// TIA Portal V20 export
DATA_BLOCK "Alarms"   // DB38
{ DB_Accessible_From_OPC_UA := 'FALSE' }
AUTHOR : ERsystem_FA2_DH. Kim
// stored: DBAccessibleFromOPCUA false, DBAccessibleFromWebserver false, MemoryReserve 100, Namespace Unit1.Em6
   VAR
      emAlarms { ExternalWritable := 'False'} : "LAF_typeAlarms";
      maintenanceFaults { ExternalWritable := 'False'} : Array[0..199] of Bool;   // PFE Maintenance Faults
      productionFaults { ExternalWritable := 'False'} : Array[0..199] of Bool;   // PFE Production Faults
      toolingFault { ExternalWritable := 'False'} : Array[0..199] of Bool;   // PFE Tooling Faults
      qualityFault { ExternalWritable := 'False'} : Array[0..199] of Bool;   // PFE Quality Faults
      throughputFaultBlocked { ExternalWritable := 'False'} : Array[0..199] of Bool;   // PFE Throughput Fault Blocked
      throughputFaultStarved { ExternalWritable := 'False'} : Array[0..199] of Bool;   // PFE Throughput Fault Starved
      throughputFault { ExternalWritable := 'False'} : Array[0..199] of Bool;   // PFE Throughput Fault
      systemFaultGeneral { ExternalWritable := 'False'} : Array[0..199] of Bool;   // PFE System Fault General
      materialFault { ExternalWritable := 'False'} : Array[0..199] of Bool;   // PFE Material Fault
      maintenanceWarnings { ExternalWritable := 'False'} : Array[0..199] of Bool;   // PFE Maintenance Warnings
      productionWarning { ExternalWritable := 'False'} : Array[0..199] of Bool;   // PFE Production Warning
      toolingWarning { ExternalWritable := 'False'} : Array[0..199] of Bool;   // PFE Tooling Warning
      qualityWarning { ExternalWritable := 'False'} : Array[0..199] of Bool;   // PFE Quality Warning
      throughputWarning { ExternalWritable := 'False'} : Array[0..199] of Bool;   // PFE Throughput Warning
      systemWarning { ExternalWritable := 'False'} : Array[0..199] of Bool;   // PFE System Warning
      materialWarning { ExternalWritable := 'False'} : Array[0..199] of Bool;   // PFE Material Warning
      maintenanceStatus { ExternalWritable := 'False'} : Array[0..199] of Bool;   // PFE Maintenance Status
      productionStatus { ExternalWritable := 'False'} : Array[0..199] of Bool;   // PFE Production Status
      toolingStatus { ExternalWritable := 'False'} : Array[0..199] of Bool;   // PFE Tooling Status
      qualityStatus { ExternalWritable := 'False'} : Array[0..199] of Bool;   // PFE Quality Status
      throughputStatus { ExternalWritable := 'False'} : Array[0..199] of Bool;   // PFE Throughput Status
      systemStatus { ExternalWritable := 'False'} : Array[0..199] of Bool;   // PFE System Status
      materialStatus { ExternalWritable := 'False'} : Array[0..199] of Bool;   // PFE Material Status
      tonMaintenanceFault { ExternalWritable := 'False'} : Array[0..199] of TON_TIME;   // PFE Maintenance Faults Ton Timer
      tonProductionFault { ExternalWritable := 'False'} : Array[0..199] of TON_TIME;   // PFE Production Faults Ton Timer
      tonToolingFault { ExternalWritable := 'False'} : Array[0..199] of TON_TIME;   // PFE Tooling Faults Ton Timer
      tonQualityFault { ExternalWritable := 'False'} : Array[0..199] of TON_TIME;   // PFE Quality Faults Ton Timer
      tonThroughputFaultBlocked { ExternalWritable := 'False'} : Array[0..199] of TON_TIME;   // PFE Throughput Fault Blocked Ton Timer
      tonThroughputFaultStarved { ExternalWritable := 'False'} : Array[0..199] of TON_TIME;   // PFE Throughput Fault Starved Ton Timer
      tonThroughputFault { ExternalWritable := 'False'} : Array[0..199] of TON_TIME;   // PFE Throughput Fault Ton Timer
      tonSystemFaultGeneral { ExternalWritable := 'False'} : Array[0..199] of TON_TIME;   // PFE System Fault General Ton Timer
      tonMaterialFault { ExternalWritable := 'False'} : Array[0..199] of TON_TIME;   // PFE Material Fault Ton Timer
      tonMaintenanceWarning { ExternalWritable := 'False'} : Array[0..199] of TON_TIME;   // PFE Maintenance Warnings Ton Timer
      tonProductionWarning { ExternalWritable := 'False'} : Array[0..199] of TON_TIME;   // PFE Production Warning Ton Timer
      tonToolingWarning { ExternalWritable := 'False'} : Array[0..199] of TON_TIME;   // PFE Tooling Warning Ton Timer
      tonQualityWarning { ExternalWritable := 'False'} : Array[0..199] of TON_TIME;   // PFE Quality Warning Ton Timer
      tonThroughputWarning { ExternalWritable := 'False'} : Array[0..199] of TON_TIME;   // PFE Throughput Warning Ton Timer
      tonSystemWarning { ExternalWritable := 'False'} : Array[0..199] of TON_TIME;   // PFE System Warning Ton Timer
      tonMaterialWarning { ExternalWritable := 'False'} : Array[0..199] of TON_TIME;   // PFE Material Warning Ton Timer
      tonMaintenanceStatus { ExternalWritable := 'False'} : Array[0..199] of TON_TIME;   // PFE Maintenance Status Ton Timer
      tonProductionStatus { ExternalWritable := 'False'} : Array[0..199] of TON_TIME;   // PFE Production Status Ton Timer
      tonToolingStatus { ExternalWritable := 'False'} : Array[0..199] of TON_TIME;   // PFE Tooling Status Ton Timer
      tonQualityStatus { ExternalWritable := 'False'} : Array[0..199] of TON_TIME;   // PFE Quality Status Ton Timer
      tonThroughputStatus { ExternalWritable := 'False'} : Array[0..199] of TON_TIME;   // PFE Throughput Status Ton Timer
      tonSystemStatus { ExternalWritable := 'False'} : Array[0..199] of TON_TIME;   // PFE System Status Ton Timer
      tonMaterialStatus { ExternalWritable := 'False'} : Array[0..199] of TON_TIME;   // PFE Material Status Ton Timer
      axisErrorCode { ExternalWritable := 'False'} : Array[0..14] of UDInt;
   END_VAR
BEGIN
   emAlarms.error := TRUE;
   emAlarms.warning := FALSE;
   emAlarms.info := FALSE;
   // maintenanceFaults[0] : FinalRoller AxisX UnSync Faults
   // maintenanceFaults[1] : StackTable OutAxisZ UnSync Faults
   // maintenanceFaults[10] : FINAL ROLLER FRONT LIMIT SENSOR(-)
   // maintenanceFaults[11] : FINAL ROLLER FRONT LIMIT SENSOR(+)
   // maintenanceFaults[12] : FINAL ROLLER REAR LIMIT SENSOR(-)
   // maintenanceFaults[13] : FINAL ROLLER REAR LIMIT SENSOR(+)
   // maintenanceFaults[14] : ANODE MANDREL FRONT Y AXIS LIMIT SENSOR(-)
   // maintenanceFaults[15] : ANODE MANDREL FRONT Y AXIS LIMIT SENSOR(+)
   // maintenanceFaults[16] : ANODE MANDREL FRONT Z AXIS LIMIT SENSOR(-)
   // maintenanceFaults[17] : ANODE MANDREL FRONT Z AXIS LIMIT SENSOR(+)
   // maintenanceFaults[18] : ANODE MANDREL REAR Y AXIS LIMIT SENSOR(-)
   // maintenanceFaults[19] : ANODE MANDREL REAR Y AXIS LIMIT SENSOR(+)
   // maintenanceFaults[20] : ANODE MANDREL REAR Z AXIS LIMIT SENSOR(-)
   // maintenanceFaults[21] : ANODE MANDREL REAR Z AXIS LIMIT SENSOR(+)
   // maintenanceFaults[22] : CATHODE MANDREL FRONT Y AXIS LIMIT SENSOR(-)
   // maintenanceFaults[23] : CATHODE MANDREL FRONT Y AXIS LIMIT SENSOR(+)
   // maintenanceFaults[24] : CATHODE MANDREL FRONT Z AXIS LIMIT SENSOR(-)
   // maintenanceFaults[25] : CATHODE MANDREL FRONT Z AXIS LIMIT SENSOR(+)
   // maintenanceFaults[26] : CATHODE MANDREL REAR Y AXIS LIMIT SENSOR(-)
   // maintenanceFaults[27] : CATHODE MANDREL REAR Y AXIS LIMIT SENSOR(+)
   // maintenanceFaults[28] : CATHODE MANDREL REAR Z AXIS LIMIT SENSOR(-)
   // maintenanceFaults[29] : CATHODE MANDREL REAR Z AXIS LIMIT SENSOR(+)
   // maintenanceFaults[30] : STACK TABLE Z-AXIS LIMIT SENSOR(-)
   // maintenanceFaults[31] : STACK TABLE Z-AXIS LIMIT SENSOR(+)
   // maintenanceFaults[32] : STACK TABLE OUT FRONT Z-AXIS LIMIT SENSOR(-)
   // maintenanceFaults[33] : STACK TABLE OUT FRONT Z-AXIS LIMIT SENSOR(+)
   // maintenanceFaults[34] : STACK TABLE OUT REAR Z-AXIS LIMIT SENSOR(-)
   // maintenanceFaults[35] : STACK TABLE OUT REAR Z-AXIS LIMIT SENSOR(+)
   // maintenanceFaults[40] : FINAL ROLLER FRONT Drive Fault
   // maintenanceFaults[41] : FINAL ROLLER REAR Drive Fault
   // maintenanceFaults[42] : ANODE MANDREL FRONT Y AXIS Drive Fault
   // maintenanceFaults[43] : ANODE MANDREL FRONT Z AXIS Drive Fault
   // maintenanceFaults[44] : ANODE MANDREL REAR Y AXIS Drive Fault
   // maintenanceFaults[45] : ANODE MANDREL REAR Z AXIS Drive Fault
   // maintenanceFaults[46] : CATHODE MANDREL FRONT Y AXIS Drive Fault
   // maintenanceFaults[47] : CATHODE MANDREL FRONT Z AXIS Drive Fault
   // maintenanceFaults[48] : CATHODE MANDREL REAR Y AXIS Drive Fault
   // maintenanceFaults[49] : CATHODE MANDREL REAR Z AXIS Drive Fault
   // maintenanceFaults[50] : STACK TABLE Z-AXIS Drive Fault
   // maintenanceFaults[51] : STACK TABLE OUT FRONT Z-AXIS Drive Fault
   // maintenanceFaults[52] : STACK TABLE OUT REAR Z-AXIS Drive Fault
   // maintenanceFaults[70] : FINAL ROLLER FRONT Home Sensor Abnomal
   // maintenanceFaults[71] : FINAL ROLLER REAR Home Sensor Abnomal
   // maintenanceFaults[72] : ANODE MANDREL FRONT Y AXIS Home Sensor Abnomal
   // maintenanceFaults[73] : ANODE MANDREL FRONT Z AXIS Home Sensor Abnomal
   // maintenanceFaults[74] : ANODE MANDREL REAR Y AXIS Home Sensor Abnomal
   // maintenanceFaults[75] : ANODE MANDREL REAR Z AXIS Home Sensor Abnomal
   // maintenanceFaults[76] : CATHODE MANDREL FRONT Y AXIS Home Sensor Abnomal
   // maintenanceFaults[77] : CATHODE MANDREL FRONT Z AXIS Home Sensor Abnomal
   // maintenanceFaults[78] : CATHODE MANDREL REAR Y AXIS Home Sensor Abnomal
   // maintenanceFaults[79] : CATHODE MANDREL REAR Z AXIS Home Sensor Abnomal
   // maintenanceFaults[80] : STACK TABLE Z-AXIS Home Sensor Abnomal
   // maintenanceFaults[81] : STACK TABLE OUT FRONT Z-AXIS Home Sensor Abnomal
   // maintenanceFaults[82] : STACK TABLE OUT REAR Z-AXIS Home Sensor Abnomal
   // productionFaults[1] : OVER COUNT of STACK
   // maintenanceWarnings[0] : FinalRoller AxisX UnSync Warnings
   // maintenanceWarnings[1] : StackTable Out AxisZ UnSync Warnings
END_DATA_BLOCK
